FUNCTION_BLOCK JackHAL_HW (* Composite Function Block Type *)
  (* Standard: 61499-2 *)
  (* Version 0.0, 9/26/2018, dmidro, nxtControl GmbH, template *)
  PACKAGE Main;
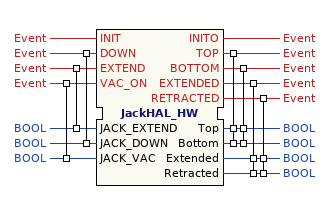
  EVENT_INPUT
    INIT; (* Initialization Request *)
    DOWN WITH JACK_DOWN;
    EXTEND WITH JACK_EXTEND;
    VAC_ON WITH JACK_VAC;
  END_EVENT
  EVENT_OUTPUT
    INITO; (* Initialization Confirm *)
    TOP WITH Top, Bottom;
    BOTTOM WITH Bottom, Top;
    EXTENDED WITH Extended, Retracted;
    RETRACTED WITH Retracted, Extended;
  END_EVENT
  VAR_INPUT
    JACK_EXTEND : BOOL; (* New value(i) for the named variable element *)
    JACK_DOWN : BOOL; (* New value(i) for the named variable element *)
    JACK_VAC : BOOL; (* New value(i) for the named variable element *)
  END_VAR
  VAR_OUTPUT
    Top : BOOL; (* Current value(i) in the named variable array element *)
    Bottom : BOOL; (* Current value(i) in the named variable array element *)
    Extended : BOOL; (* Current value(i) in the named variable array element *)
    Retracted : BOOL; (* Current value(i) in the named variable array element *)
  END_VAR
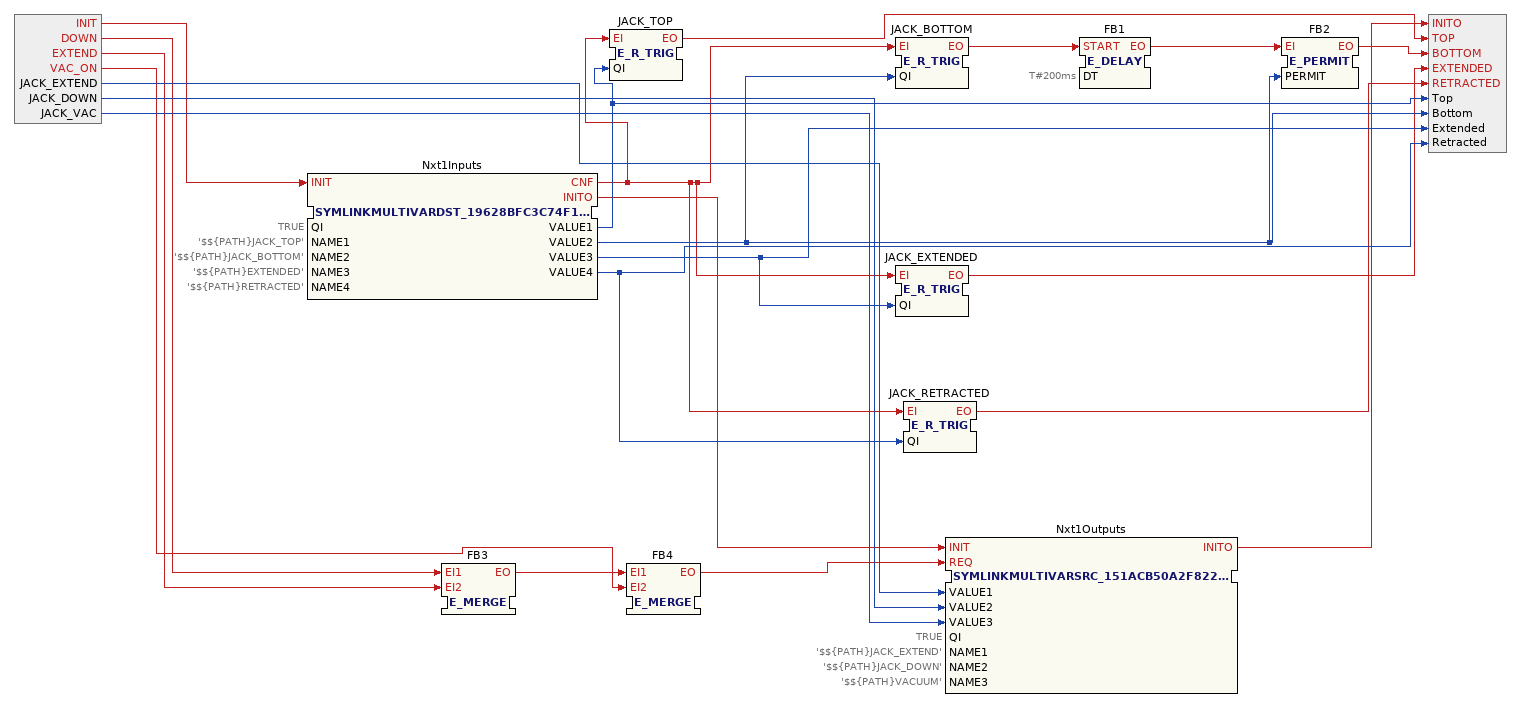
  FBS
    Nxt1Inputs : SYMLINKMULTIVARDST_19628BFC3C74F1AB1(QI := TRUE, NAME1 := '$${PATH}JACK_TOP', NAME2 := '$${PATH}JACK_BOTTOM', NAME3 := '$${PATH}EXTENDED', NAME4 := '$${PATH}RETRACTED'); {SET_ATTRIBUTE(Configuration.GenericFBType.InterfaceParams, Runtime.System#I:=4;VALUE${I$}:BOOL,BOOL,BOOL,BOOL)}
    Nxt1Outputs : SYMLINKMULTIVARSRC_151ACB50A2F8223B2(QI := TRUE, NAME1 := '$${PATH}JACK_EXTEND', NAME2 := '$${PATH}JACK_DOWN', NAME3 := '$${PATH}VACUUM'); {SET_ATTRIBUTE(Configuration.GenericFBType.InterfaceParams, Runtime.System#I:=3;VALUE${I$}:BOOL,BOOL,BOOL)}
    JACK_EXTENDED : E_R_TRIG;
    JACK_RETRACTED : E_R_TRIG;
    JACK_TOP : E_R_TRIG;
    JACK_BOTTOM : E_R_TRIG;
    FB1 : E_DELAY(DT := T#200ms);
    FB2 : E_PERMIT;
    FB3 : E_MERGE;
    FB4 : E_MERGE;
  END_FBS
  EVENT_CONNECTIONS
    JACK_EXTENDED.EO TO EXTENDED;
    JACK_RETRACTED.EO TO RETRACTED;
    JACK_TOP.EO TO TOP;
    JACK_BOTTOM.EO TO FB1.START;
    FB1.EO TO FB2.EI;
    FB2.EO TO BOTTOM;
    FB3.EO TO FB4.EI1;
    VAC_ON TO FB4.EI2;
    DOWN TO FB3.EI1;
    EXTEND TO FB3.EI2;
    INIT TO Nxt1Inputs.INIT;
    Nxt1Inputs.CNF TO JACK_RETRACTED.EI;
    Nxt1Inputs.CNF TO JACK_EXTENDED.EI;
    Nxt1Inputs.CNF TO JACK_TOP.EI;
    Nxt1Inputs.CNF TO JACK_BOTTOM.EI;
    Nxt1Inputs.INITO TO Nxt1Outputs.INIT;
    FB4.EO TO Nxt1Outputs.REQ;
    Nxt1Outputs.INITO TO INITO;
  END_CONNECTIONS
  DATA_CONNECTIONS
    Nxt1Inputs.VALUE1 TO JACK_TOP.QI;
    Nxt1Inputs.VALUE2 TO JACK_BOTTOM.QI;
    Nxt1Inputs.VALUE2 TO FB2.PERMIT;
    Nxt1Inputs.VALUE3 TO JACK_EXTENDED.QI;
    Nxt1Inputs.VALUE4 TO JACK_RETRACTED.QI;
    JACK_EXTEND TO Nxt1Outputs.VALUE1;
    JACK_DOWN TO Nxt1Outputs.VALUE2;
    JACK_VAC TO Nxt1Outputs.VALUE3;
    Nxt1Inputs.VALUE1 TO Top;
    Nxt1Inputs.VALUE2 TO Bottom;
    Nxt1Inputs.VALUE3 TO Extended;
    Nxt1Inputs.VALUE4 TO Retracted;
  END_CONNECTIONS
END_FUNCTION_BLOCK
